(* IEC 61131-3 sources: cds-text-sync-reference-project/project-view/CODESYS_Linux_SL/PLC Logic/CI_CD_Application, 6 files *)

(* ---- FB_Arithmetic.st ---- *)
FUNCTION_BLOCK FB_Arithmetic
VAR_INPUT
	rA : REAL;
	rB : REAL;
	eOp : USINT; // 0=Add, 1=Sub, 2=Mul, 3=Div
	xExecute : BOOL;
END_VAR
VAR_OUTPUT
	rResult : REAL;
	xDone : BOOL;
END_VAR
VAR
	xPrev : BOOL;
END_VAR

// --- implementation ---

IF xExecute AND NOT xPrev THEN
	CASE eOp OF
		0: rResult := rA + rB;
		1: rResult := rA - rB;
		2: rResult := rA * rB;
		3:
			IF rB <> 0.0 THEN
				rResult := rA / rB;
			ELSE
				rResult := 0.0;
			END_IF
		ELSE
			rResult := 0.0;
	END_CASE
	xDone := TRUE;
END_IF

IF NOT xExecute THEN
	xDone := FALSE;
END_IF

xPrev := xExecute;

(* ---- FB_Checksum.st ---- *)
FUNCTION_BLOCK FB_Checksum
VAR_INPUT
	bA : BYTE;
	bB : BYTE;
	bC : BYTE;
	xExecute : BOOL;
END_VAR
VAR_OUTPUT
	bResult : BYTE;
	xDone : BOOL;
END_VAR
VAR
	xPrev : BOOL;
END_VAR

// --- implementation ---

IF xExecute AND NOT xPrev THEN
	bResult := bA XOR bB XOR bC;
	xDone := TRUE;
END_IF

IF NOT xExecute THEN
	xDone := FALSE;
END_IF

xPrev := xExecute;

(* ---- FB_Deadband.st ---- *)
FUNCTION_BLOCK FB_Deadband
VAR_INPUT
	rValue : REAL;
	rBand : REAL;
	xExecute : BOOL;
END_VAR
VAR_OUTPUT
	rResult : REAL;
	xDone : BOOL;
END_VAR
VAR
	xPrev : BOOL;
END_VAR

// --- implementation ---

IF xExecute AND NOT xPrev THEN
	IF rValue > -rBand AND rValue < rBand THEN
		rResult := 0.0;
	ELSE
		rResult := rValue;
	END_IF
	xDone := TRUE;
END_IF

IF NOT xExecute THEN
	xDone := FALSE;
END_IF

xPrev := xExecute;

(* ---- FB_RangeCheck.st ---- *)
FUNCTION_BLOCK FB_RangeCheck
VAR_INPUT
	rValue : REAL;
	rMin : REAL;
	rMax : REAL;
	xExecute : BOOL;
END_VAR
VAR_OUTPUT
	xInRange : BOOL;
	xDone : BOOL;
END_VAR

// --- implementation ---

IF xExecute THEN
	xInRange := rValue >= rMin AND rValue <= rMax;
	xDone := TRUE;
ELSE
	xDone := FALSE;
	xInRange := FALSE;
END_IF

(* ---- FB_Scale.st ---- *)
FUNCTION_BLOCK FB_Scale
VAR_INPUT
	rRaw : REAL;
	rRawMin : REAL;
	rRawMax : REAL;
	rScaledMin : REAL;
	rScaledMax : REAL;
	xExecute : BOOL;
END_VAR
VAR_OUTPUT
	rResult : REAL;
	xDone : BOOL;
	xError : BOOL;
END_VAR

// --- implementation ---

IF xExecute THEN
	IF rRawMax <> rRawMin THEN
		xError := FALSE;
		rResult := rScaledMin + (rRaw - rRawMin) / (rRawMax - rRawMin) * (rScaledMax - rScaledMin);

		// Clamp (handle both normal and reversed scaled ranges)
		IF rResult < rScaledMin THEN rResult := rScaledMin; END_IF
		IF rResult > rScaledMax THEN rResult := rScaledMax; END_IF
	ELSE
		rResult := rScaledMin;
		xError   := TRUE;
	END_IF

	xDone := TRUE;
ELSE
	xDone  := FALSE;
	xError := FALSE;
END_IF

(* ---- MAIN.st ---- *)
PROGRAM MAIN
VAR
	// CI/CD test instances â variables visible via read_variable/write_variable
	fbArith : FB_Arithmetic;
	fbScale : FB_Scale;
	fbDeadband : FB_Deadband;
	fbRangeCheck : FB_RangeCheck;
	fbChecksum : FB_Checksum;
	fbCounter : FB_Counter_UD;
END_VAR

// --- implementation ---

// Pass-through call: inputs read from instance variables (set via online API),
// outputs written back to instance variables.
fbArith(rA := fbArith.rA, rB := fbArith.rB,
        eOp := fbArith.eOp, xExecute := fbArith.xExecute);

fbScale(rRaw := fbScale.rRaw, rRawMin := fbScale.rRawMin,
        rRawMax := fbScale.rRawMax, rScaledMin := fbScale.rScaledMin,
        rScaledMax := fbScale.rScaledMax, xExecute := fbScale.xExecute);

fbDeadband(rValue := fbDeadband.rValue, rBand := fbDeadband.rBand,
           xExecute := fbDeadband.xExecute);

fbRangeCheck(rValue := fbRangeCheck.rValue, rMin := fbRangeCheck.rMin,
             rMax := fbRangeCheck.rMax, xExecute := fbRangeCheck.xExecute);

fbChecksum(bA := fbChecksum.bA, bB := fbChecksum.bB,
           bC := fbChecksum.bC, xExecute := fbChecksum.xExecute);

fbCounter(xUp := fbCounter.xUp, xDown := fbCounter.xDown,
          xReset := fbCounter.xReset, uiLimit := fbCounter.uiLimit);
